// TIA Portal V16 export
// export: Created 2021-08-30T11:09:31.4670215Z, ExportSetting WithDefaults, DisplayName Totally Integrated Automation Portal, DisplayVersion V16 Update 3, DisplayName TIA Portal Version Control Interface, DisplayVersion V16 Update 2, DisplayName TIA Portal Openness, DisplayVersion V16 Update 3, DisplayName TIA Portal Teamcenter Gateway, DisplayVersion V16, DisplayName STEP 7 Professional, DisplayVersion V16 Update 3, DisplayName STEP 7 Safety, DisplayVersion V16, DisplayName WinCC Advanced, DisplayVersion V16 Update 3
FUNCTION_BLOCK "hardwareTimePulse"   // FB12, FBD
{ S7_Optimized_Access := 'FALSE' }
VERSION : 0.1
// stored: AutoNumber false, IsIECCheckEnabled false, SetENOAutomatically false, UDAEnableTagReadback false
   VAR DB_SPECIFIC
      pTrig1HZ : Bool;
      pTrig05Hz : Bool;
      pTrig0625Hz : Bool;
      pTrig1_25HZ : Bool;
      pTrig2HZ : Bool;
      pTrig2_5Hz : Bool;
      pTirg5Hz : Bool;
      pTrig10Hz : Bool;
   END_VAR
   VAR_TEMP   // added for the SCL form of the ladder/FBD networks
      _w1 : Bool;
   END_VAR
BEGIN

REGION Network 1
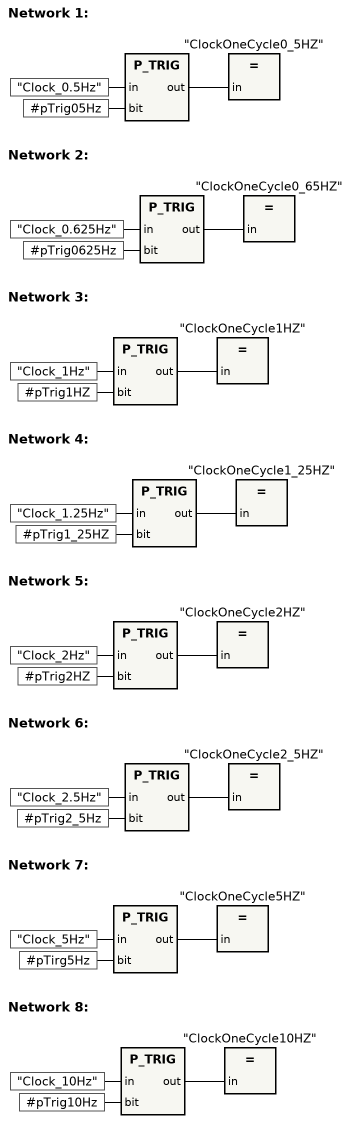
   #_w1 := "Clock_0.5Hz" AND NOT #pTrig05Hz;   // rising edge
   #pTrig05Hz := "Clock_0.5Hz";
   "ClockOneCycle0_5HZ" := #_w1;
END_REGION

REGION Network 2
   #_w1 := "Clock_0.625Hz" AND NOT #pTrig0625Hz;   // rising edge
   #pTrig0625Hz := "Clock_0.625Hz";
   "ClockOneCycle0_65HZ" := #_w1;
END_REGION

REGION Network 3
   #_w1 := "Clock_1Hz" AND NOT #pTrig1HZ;   // rising edge
   #pTrig1HZ := "Clock_1Hz";
   "ClockOneCycle1HZ" := #_w1;
END_REGION

REGION Network 4
   #_w1 := "Clock_1.25Hz" AND NOT #pTrig1_25HZ;   // rising edge
   #pTrig1_25HZ := "Clock_1.25Hz";
   "ClockOneCycle1_25HZ" := #_w1;
END_REGION

REGION Network 5
   #_w1 := "Clock_2Hz" AND NOT #pTrig2HZ;   // rising edge
   #pTrig2HZ := "Clock_2Hz";
   "ClockOneCycle2HZ" := #_w1;
END_REGION

REGION Network 6
   #_w1 := "Clock_2.5Hz" AND NOT #pTrig2_5Hz;   // rising edge
   #pTrig2_5Hz := "Clock_2.5Hz";
   "ClockOneCycle2_5HZ" := #_w1;
END_REGION

REGION Network 7
   #_w1 := "Clock_5Hz" AND NOT #pTirg5Hz;   // rising edge
   #pTirg5Hz := "Clock_5Hz";
   "ClockOneCycle5HZ" := #_w1;
END_REGION

REGION Network 8
   #_w1 := "Clock_10Hz" AND NOT #pTrig10Hz;   // rising edge
   #pTrig10Hz := "Clock_10Hz";
   "ClockOneCycle10HZ" := #_w1;
END_REGION
END_FUNCTION_BLOCK
